FUNCTION_BLOCK SkillSwing (* Basic Function Block Type *)
  (* Standard: 61499-2 *)
  (* Version 0.0, 12/05/2025, autogen, Swing skill: arm moves left and right twice *)
  PACKAGE Main;
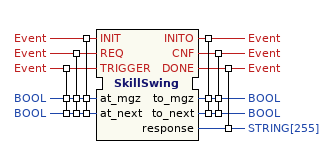
  EVENT_INPUT
    INIT WITH at_mgz, at_next; (* Initialization Request *)
    REQ WITH at_mgz, at_next; (* Normal Execution Request *)
    TRIGGER WITH at_mgz, at_next;
  END_EVENT
  EVENT_OUTPUT
    INITO WITH to_mgz, to_next; (* Initialization Confirm *)
    CNF WITH to_mgz, to_next; (* Execution Confirmation *)
    DONE WITH response;
  END_EVENT
  VAR_INPUT
    at_mgz : BOOL;
    at_next : BOOL;
  END_VAR
  VAR_OUTPUT
    to_mgz : BOOL;
    to_next : BOOL;
    response : STRING[255];
  END_VAR
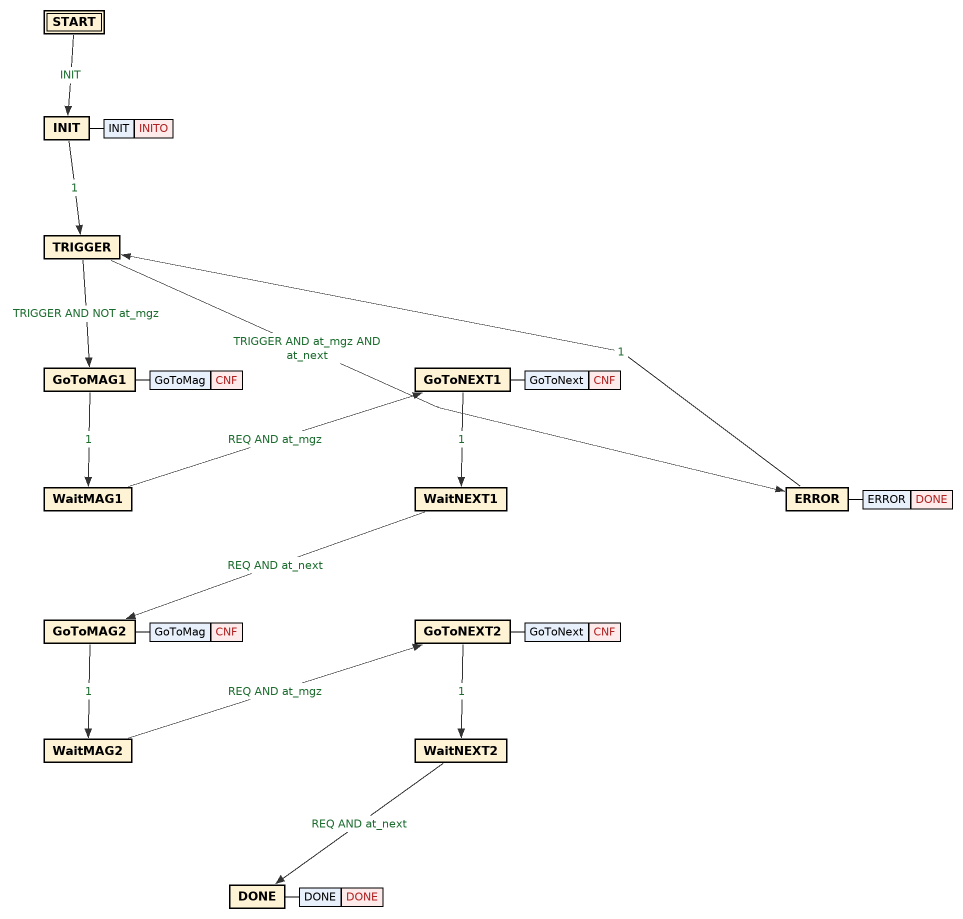
  EC_STATES
    START; (* Initial State *)
    INIT : INIT -> INITO; (* Initialization *)
    TRIGGER;
    GoToMAG1 : GoToMag -> CNF;
    WaitMAG1;
    GoToNEXT1 : GoToNext -> CNF;
    WaitNEXT1;
    GoToMAG2 : GoToMag -> CNF;
    WaitMAG2;
    GoToNEXT2 : GoToNext -> CNF;
    WaitNEXT2;
    DONE : DONE -> DONE;
    ERROR : ERROR -> DONE;
  END_STATES
  EC_TRANSITIONS
    START TO INIT := INIT;
    INIT TO TRIGGER := 1;
    TRIGGER TO GoToMAG1 := TRIGGER AND NOT at_mgz;
    TRIGGER TO ERROR := TRIGGER AND at_mgz AND at_next;
    GoToMAG1 TO WaitMAG1 := 1;
    WaitMAG1 TO GoToNEXT1 := REQ AND at_mgz;
    GoToNEXT1 TO WaitNEXT1 := 1;
    WaitNEXT1 TO GoToMAG2 := REQ AND at_next;
    GoToMAG2 TO WaitMAG2 := 1;
    WaitMAG2 TO GoToNEXT2 := REQ AND at_mgz;
    GoToNEXT2 TO WaitNEXT2 := 1;
    WaitNEXT2 TO DONE := REQ AND at_next;
    ERROR TO TRIGGER := 1;
  END_TRANSITIONS
  ALGORITHM INIT IN ST: (* Initialization algorithm *)
to_mgz := FALSE;
to_next := FALSE;
response := 'INITIALISED';
  END_ALGORITHM
  ALGORITHM GoToMag IN ST:
to_mgz := TRUE;
to_next := FALSE;
  END_ALGORITHM
  ALGORITHM GoToNext IN ST:
to_mgz := FALSE;
to_next := TRUE;
  END_ALGORITHM
  ALGORITHM DONE IN ST:
response := 'SWING COMPLETED';
TRIGGER := FALSE;
  END_ALGORITHM
  ALGORITHM ERROR IN ST:
response := 'ERROR: ALREADY AT POSITION';
TRIGGER := FALSE;
  END_ALGORITHM
END_FUNCTION_BLOCK
(* other elements stored in the file *)
(* Transitions *)
(* Sequence: TRIGGER -> GoToMAG1 (if not at_mgz) or ERROR if already *)
(* After commanding, wait for confirmation: REQ and at_mgz *)
